(* IEC 61131-3 sources: beeguard/archive, 2 files *)

(* ---- analog.st ---- *)
FUNCTION_BLOCK AOI_CM_AIN
VAR_INPUT
	IN_IOH: BOOL;
	IN_INH1: DINT;
	IN_OVR: BOOL;
	IN_UNR: BOOL;
	IN_RAW: REAL;
	CMD_ALM_RES: BOOL;
	IN_CLOCK: DT;	// CURRENT DATE AND TIME, PASSED TO THE ALARMS FOR TIME STAMPS
END_VAR
VAR_INPUT PERSISTENT RETAIN
	CFG_EN: BOOL;
	CFG_RU_MAX: DINT;
	CFG_RU_MIN: DINT;
	CFG_EU_MAX: REAL;
	CFG_EU_MIN: REAL;
	CFG_HIHI_SP: REAL;
	CFG_HI_SP: REAL;
	CFG_LO_SP: REAL;
	CFG_LOLO_SP: REAL;
	CFG_FRZN_SP: REAL;
	CFG_DEC_PT: DINT;
	CFG_DESC: STRING;
	CFG_DEV_TYPE: DINT;
	CFG_EID: STRING;
	CFG_EN_ALM_HI: BOOL;
	CFG_EN_ALM_HIHI: BOOL;
	CFG_EN_ALM_IOH: BOOL;
	CFG_EN_ALM_LO: BOOL;
	CFG_EN_ALM_LOLO: BOOL;
	CFG_EN_ALM_OOR: BOOL;
	CFG_EN_ALM_FRZN: BOOL;
	CFG_EN_IOH: BOOL;
	CFG_EN_OOR: BOOL;
	CFG_EN_SCL: BOOL;
	CFG_EN_TOT: BOOL;
	CFG_EN_FRZN: BOOL;
	CFG_HI_DT: DINT;
	CFG_HIHI_DT: DINT;
	CFG_LO_DT: DINT;
	CFG_LOLO_DT: DINT;
	CFG_OOR_DT: DINT;
	CFG_FRZN_DT: DINT;
	CFG_SCL_TYP: DINT;
	CFG_UNITS: STRING;
	SIM: BOOL;
	CFG_TMR_DISABLE_SIM: BOOL;
END_VAR
VAR_IN_OUT
	ALMD_HIHI: BG_ALM_DIG;
	ALMD_HI: BG_ALM_DIG;
	ALMD_LO: BG_ALM_DIG;
	ALMD_LOLO: BG_ALM_DIG;
	ALMD_OOR: BG_ALM_DIG;
	ALMD_IOH: BG_ALM_DIG;
	ALMD_FRZN: BG_ALM_DIG;
END_VAR
VAR_OUTPUT
	STS_RDY2GO: BOOL;
	VAL_ACT: REAL;
	ALM_HIHI: BOOL;
	ALM_HI: BOOL;
	ALM_LO: BOOL;
	ALM_LOLO: BOOL;
	ALM_OOR: BOOL;
	ALM_IOH: BOOL;
	ALM_FRZN: BOOL;
	STS_HIHI: BOOL;
	STS_HI: BOOL;
	STS_LO: BOOL;
	STS_LOLO: BOOL;
	STS_OOR: BOOL;
	STS_IOH: BOOL;
	STS_FRZN: BOOL;
	CFG_VERSION: REAL;
	STS_ALM_ANY: BOOL;
	STS_ALM_ANY_UNACK: BOOL;
	ALM_ANY: BOOL;
	VAL_S: DINT;
END_VAR
VAR
	SIM_ONS: R_TRIG;
	WRK_B0: BOOL;
	WRK_B1: BOOL;
	WRK_ONS: ARRAY[0..15] OF R_TRIG;
	WRK_R: ARRAY[0..6] OF REAL;
	WRK_T: ARRAY[0..7] OF TON;
END_VAR

(*===========================================================================
AOI: CM_AIN
Date Last Updated: 5-27-2024
===========================================================================*)
//CFG_VERSION:= 1.0; // ORIGINAL
//CFG_VERSION := 2.0; //ADDED THE DIGITAL ALARM FUNCTION BLOCK
//CFG_VERSION := 2.1; //ADDED FRONZEN DATA ALARM LOGIC
//CFG_VERSION := 2.2; //DIGITAL ALARM 3.0: ACK+RESET, CLOCK, INHIBIT = SUPPRESS, SINGLE ON-DELAY, IOH INHIBIT ON BIT 6
CFG_VERSION := 2.3; //USES BG_ALM_DIG 3.1 NAMES; CLOCK INPUT RENAMED IN_CLOCK
(*===========================================================================
RETURN IF DISABLED  - If Module is Disabled, Scan One Last Time for Cleanup, Then Return
===========================================================================*)
IF NOT(CFG_EN) THEN
	WRK_ONS[1].CLK := TRUE;
	IF WRK_ONS[1].Q THEN
		WRK_B1 := TRUE;
	END_IF
	IF NOT(WRK_B1) THEN
		JMP EXIT_AOI_CM_AIN;
	END_IF
ELSE
	WRK_B1 := FALSE;
	WRK_ONS[1].CLK := FALSE;
END_IF

(*===========================================================================
SETUP - Clean up the Config: Enable Alarming depending on what Inputs are Confirmed in the System.
===========================================================================*)
IF NOT(CFG_EN_IOH) THEN
	CFG_EN_ALM_IOH := FALSE;
END_IF
IF NOT(CFG_EN_OOR) THEN
	CFG_EN_ALM_OOR := FALSE;
END_IF
IF NOT(CFG_EN_FRZN) THEN
	CFG_EN_ALM_FRZN := FALSE;
END_IF
(*===========================================================================
SETUP - Prevent wire-framing in HMI during start up (this prevents dividing by zero).
===========================================================================*)
IF CFG_EU_MAX = 0.0 THEN
	CFG_EU_MAX := 100;
END_IF

(*===========================================================================
TIMER PRESETS - Check and correct for invalid Timer Preset values
===========================================================================*)
WRK_T[1].PT := DINT_TO_TIME(ABS(CFG_HIHI_DT)*1000);
WRK_T[2].PT := DINT_TO_TIME(ABS(CFG_HI_DT)*1000);
WRK_T[3].PT := DINT_TO_TIME(ABS(CFG_LO_DT)*1000);
WRK_T[4].PT := DINT_TO_TIME(ABS(CFG_LOLO_DT)*1000);
WRK_T[5].PT := DINT_TO_TIME(ABS(CFG_OOR_DT)*1000);
WRK_T[7].PT := DINT_TO_TIME(ABS(CFG_FRZN_DT)*1000);

(*===========================================================================
COMMANDS - Latch Internal Work Bit To Clear All Alarms
===========================================================================*)
SIM_ONS.CLK := SIM;
IF CMD_ALM_RES OR (SIM_ONS.Q) THEN
	WRK_B0 := TRUE;
	CMD_ALM_RES := FALSE;
END_IF

(*===========================================================================
STATUS - I/O Health
===========================================================================*)
IF (CFG_EN_IOH AND IN_IOH) OR (NOT(CFG_EN_IOH)) OR (SIM) THEN
	STS_IOH := TRUE;
ELSE
	STS_IOH := FALSE;
END_IF

(*===========================================================================
STATUS - I/O Health
===========================================================================*)
IF (CFG_EN_OOR) AND (IN_OVR OR IN_UNR) THEN
	STS_OOR := TRUE;
ELSE
	STS_OOR := FALSE;
END_IF

(*===========================================================================
STATUS  - CM Ready to Go
CM is Ready to Go if it is Enabled, it's HOA(s) are in the Auto position and Interlocks are met.
NOTE: Not all conditions may exist for a given CM Cla
===========================================================================*)
IF (CFG_EN AND STS_IOH) THEN
	STS_RDY2GO := TRUE;
ELSE
	STS_RDY2GO := FALSE;
END_IF

(*===========================================================================
ALARMS HIHI - Determine HIHI Alarm if Alarms are Enabled.  If an Alarm is already
present when it is Disabled becomes it will stay TRUE.
===========================================================================*)
IF (VAL_ACT > CFG_HIHI_SP) THEN
	WRK_T[1](IN := TRUE);
	IF WRK_T[1].Q THEN
		STS_HIHI := TRUE;
		IF NOT(IN_INH1.0) AND CFG_EN_ALM_HIHI THEN
			ALM_HIHI := TRUE;
		ELSE
			ALM_HIHI := FALSE;
		END_IF
	ELSE
		STS_HIHI := FALSE;
	END_IF
ELSE
	STS_HIHI := FALSE;
	ALM_HIHI := FALSE;
	WRK_T[1](IN := FALSE);
END_IF

// INHIBIT SUPPRESSES THE ALARM INSTEAD OF RETURNING IT TO NORMAL. WRK_T[1] IS THE ONLY ON-DELAY.
ALMD_HIHI(IN_SIGNAL := CFG_EN_ALM_HIHI AND STS_HIHI, CMD_PG_SUPPRESS := IN_INH1.0, CMD_PG_UNSUPPRESS := NOT(IN_INH1.0),
	CFG_ACK_REQ := TRUE, CFG_LATCH := TRUE, CFG_ON_DELAY_MS := 0, IN_CLOCK := IN_CLOCK);

IF WRK_B0 THEN
	 WRK_ONS[5].CLK := TRUE;
	 IF WRK_ONS[5].Q THEN
		 ALMD_HIHI.CMD_OP_ACK := TRUE;
		 ALMD_HIHI.CMD_OP_RESET := TRUE;
	 END_IF
ELSE
	WRK_ONS[5].CLK := FALSE;
END_IF

(*===========================================================================
ALARMS HI - Determine HI Alarm if Alarms are Enabled.  If an Alarm is already
present when it is Disabled becomes it will stay TRUE.
===========================================================================*)
IF (VAL_ACT > CFG_HI_SP) THEN
	WRK_T[2](IN := TRUE);
	IF WRK_T[2].Q THEN
		STS_HI := TRUE;
		IF NOT(IN_INH1.1) AND CFG_EN_ALM_HI THEN
			ALM_HI := TRUE;
		ELSE
			ALM_HI := FALSE;
		END_IF
	ELSE
		STS_HI := FALSE;
	END_IF
ELSE
	STS_HI := FALSE;
	ALM_HI := FALSE;
	WRK_T[2](IN := FALSE);
END_IF

ALMD_HI(IN_SIGNAL := CFG_EN_ALM_HI AND STS_HI, CMD_PG_SUPPRESS := IN_INH1.1, CMD_PG_UNSUPPRESS := NOT(IN_INH1.1),
	CFG_ACK_REQ := TRUE, CFG_LATCH := TRUE, CFG_ON_DELAY_MS := 0, IN_CLOCK := IN_CLOCK);

IF WRK_B0 THEN
	 WRK_ONS[7].CLK := TRUE;
	 IF WRK_ONS[7].Q THEN
		 ALMD_HI.CMD_OP_ACK := TRUE;
		 ALMD_HI.CMD_OP_RESET := TRUE;
	 END_IF
ELSE
	WRK_ONS[7].CLK := FALSE;
END_IF

(*===========================================================================
ALARMS LO - Determine LO Alarm if Alarms are Enabled.  If an Alarm is already
present when it is Disabled becomes it will stay TRUE.
===========================================================================*)
IF (VAL_ACT < CFG_LO_SP) THEN
	WRK_T[3](IN := TRUE);
	IF WRK_T[3].Q THEN
		STS_LO := TRUE;
		IF NOT(IN_INH1.2) AND CFG_EN_ALM_LO THEN
			ALM_LO := TRUE;
		ELSE
			ALM_LO := FALSE;
		END_IF
	ELSE
		STS_LO := FALSE;
	END_IF
ELSE
	STS_LO := FALSE;
	ALM_LO := FALSE;
	WRK_T[3](IN := FALSE);
END_IF

ALMD_LO(IN_SIGNAL := CFG_EN_ALM_LO AND STS_LO, CMD_PG_SUPPRESS := IN_INH1.2, CMD_PG_UNSUPPRESS := NOT(IN_INH1.2),
	CFG_ACK_REQ := TRUE, CFG_LATCH := TRUE, CFG_ON_DELAY_MS := 0, IN_CLOCK := IN_CLOCK);

IF WRK_B0 THEN
	 WRK_ONS[9].CLK := TRUE;
	 IF WRK_ONS[9].Q THEN
		 ALMD_LO.CMD_OP_ACK := TRUE;
		 ALMD_LO.CMD_OP_RESET := TRUE;
	 END_IF
ELSE
	WRK_ONS[9].CLK := FALSE;
END_IF

(*===========================================================================
ALARMS LOLO - Determine LOLO Alarm if Alarms are Enabled.  If an Alarm is already
present when it is Disabled becomes it will stay TRUE.
===========================================================================*)
IF (VAL_ACT < CFG_LOLO_SP) THEN
	WRK_T[4](IN := TRUE);
	IF WRK_T[4].Q THEN
		STS_LOLO := TRUE;
		IF NOT(IN_INH1.3) AND CFG_EN_ALM_LOLO THEN
			ALM_LOLO := TRUE;
		ELSE
			ALM_LOLO := FALSE;
		END_IF
	ELSE
		STS_LOLO := FALSE;
	END_IF
ELSE
	STS_LOLO := FALSE;
	ALM_LOLO := FALSE;
	WRK_T[4](IN := FALSE);
END_IF

ALMD_LOLO(IN_SIGNAL := CFG_EN_ALM_LOLO AND STS_LOLO, CMD_PG_SUPPRESS := IN_INH1.3, CMD_PG_UNSUPPRESS := NOT(IN_INH1.3),
	CFG_ACK_REQ := TRUE, CFG_LATCH := TRUE, CFG_ON_DELAY_MS := 0, IN_CLOCK := IN_CLOCK);

IF WRK_B0 THEN
	 WRK_ONS[11].CLK := TRUE;
	 IF WRK_ONS[11].Q THEN
		 ALMD_LOLO.CMD_OP_ACK := TRUE;
		 ALMD_LOLO.CMD_OP_RESET := TRUE;
	 END_IF
ELSE
	WRK_ONS[11].CLK := FALSE;
END_IF

(*===========================================================================
ALARMS - Out of Range
===========================================================================*)
IF (CFG_EN_ALM_OOR AND STS_OOR) THEN
	WRK_T[5](IN := TRUE);
	IF WRK_T[5].Q THEN
		//STS_OOR := TRUE; SEE LINE 35
		IF NOT(IN_INH1.4) THEN
			ALM_OOR := TRUE;
		ELSE
			ALM_OOR := FALSE;
		END_IF
	END_IF
ELSE
	ALM_OOR := FALSE;
	WRK_T[5](IN := FALSE);
END_IF

ALMD_OOR(IN_SIGNAL := CFG_EN_ALM_OOR AND STS_OOR AND WRK_T[5].Q, CMD_PG_SUPPRESS := IN_INH1.4, CMD_PG_UNSUPPRESS := NOT(IN_INH1.4),
	CFG_ACK_REQ := TRUE, CFG_LATCH := TRUE, CFG_ON_DELAY_MS := 0, IN_CLOCK := IN_CLOCK);

IF WRK_B0 THEN
	 WRK_ONS[13].CLK := TRUE;
	 IF WRK_ONS[13].Q THEN
		 ALMD_OOR.CMD_OP_ACK := TRUE;
		 ALMD_OOR.CMD_OP_RESET := TRUE;
	 END_IF
ELSE
	WRK_ONS[13].CLK := FALSE;
END_IF

(*===========================================================================
ALARMS - FROZEN VALUE
===========================================================================*)
IF (VAL_ACT = CFG_FRZN_SP) THEN
	STS_FRZN := TRUE;
ELSE
	STS_FRZN := FALSE;
END_IF

IF (CFG_EN_ALM_FRZN AND STS_FRZN) THEN
	WRK_T[7](IN := TRUE);
	IF WRK_T[7].Q THEN
		//STS_FRZN := TRUE; SEE LINE 35
		IF NOT(IN_INH1.5)THEN
			ALM_FRZN := TRUE;
		ELSE
			ALM_FRZN := FALSE;
		END_IF
	END_IF
ELSE
	ALM_FRZN := FALSE;
	WRK_T[7](IN := FALSE);
END_IF

IF WRK_T[7].ET > T#0S OR CFG_EN_ALM_FRZN THEN
	CFG_FRZN_SP := VAL_ACT;
END_IF

// CFG_FRZN_DT IS NOW THE ONLY FROZEN DELAY (THE EXTRA 60 S IN THE ALARM BLOCK WAS REMOVED).
ALMD_FRZN(IN_SIGNAL := CFG_EN_ALM_FRZN AND STS_FRZN AND WRK_T[7].Q, CMD_PG_SUPPRESS := IN_INH1.5, CMD_PG_UNSUPPRESS := NOT(IN_INH1.5),
	CFG_ACK_REQ := TRUE, CFG_LATCH := TRUE, CFG_ON_DELAY_MS := 0, IN_CLOCK := IN_CLOCK);

IF WRK_B0 THEN
	 WRK_ONS[14].CLK := TRUE;
	 IF WRK_ONS[14].Q THEN
		 ALMD_FRZN.CMD_OP_ACK := TRUE;
		 ALMD_FRZN.CMD_OP_RESET := TRUE;
	 END_IF
ELSE
	WRK_ONS[14].CLK := FALSE;
END_IF

(*===========================================================================
ALARM - I/O Health (Includes Module Health, Channel Calibration Fault, or Channel Fault Alarms)
===========================================================================*)
// I/O HEALTH HAS ITS OWN INHIBIT BIT 6 (IT SHARED BIT 5 WITH FROZEN VALUE).
// IT HAS NO OTHER DELAY, SO IT KEEPS THE 1 S ON-DELAY IN THE ALARM BLOCK.
IF CFG_EN_ALM_IOH AND NOT(STS_IOH) AND NOT(IN_INH1.6) THEN
	ALM_IOH := TRUE;
ELSE
	ALM_IOH := FALSE;
END_IF

ALMD_IOH(IN_SIGNAL := CFG_EN_ALM_IOH AND NOT(STS_IOH), CMD_PG_SUPPRESS := IN_INH1.6, CMD_PG_UNSUPPRESS := NOT(IN_INH1.6),
	CFG_ACK_REQ := TRUE, CFG_LATCH := TRUE, CFG_ON_DELAY_MS := 1000, IN_CLOCK := IN_CLOCK);

IF WRK_B0 THEN
	 WRK_ONS[15].CLK := TRUE;
	 IF WRK_ONS[15].Q THEN
		 ALMD_IOH.CMD_OP_ACK := TRUE;
		 ALMD_IOH.CMD_OP_RESET := TRUE;
	 END_IF
ELSE
	WRK_ONS[15].CLK := FALSE;
END_IF

(*===========================================================================
ALARMS - Any Alarm
===========================================================================*)
IF ALM_HIHI OR ALM_HI OR ALM_LO OR ALM_LOLO OR ALM_OOR OR ALM_IOH OR ALM_FRZN THEN
	ALM_ANY := TRUE;
	STS_ALM_ANY := TRUE;
ELSE
	ALM_ANY := FALSE;
	STS_ALM_ANY := FALSE;
END_IF

(*===========================================================================
ALARMS - Check to see if there are any unacknowledged alarms, including latched
alarms whose condition has already cleared.
===========================================================================*)
IF ALMD_HIHI.STS_UNACKED OR ALMD_HI.STS_UNACKED OR ALMD_LO.STS_UNACKED OR ALMD_LOLO.STS_UNACKED OR ALMD_OOR.STS_UNACKED OR ALMD_IOH.STS_UNACKED OR ALMD_FRZN.STS_UNACKED THEN
	STS_ALM_ANY_UNACK := TRUE;
ELSE
	STS_ALM_ANY_UNACK := FALSE;
END_IF

(*===========================================================================
VALUES - State (HMI Color)
0 = Normal
1 = In Alarm
2 = Disabled
===========================================================================*)
IF NOT ALM_ANY THEN
	VAL_S := 0;
END_IF
IF ALM_ANY AND STS_ALM_ANY_UNACK THEN
	VAL_S := 1;
END_IF
IF ALM_ANY AND NOT STS_ALM_ANY_UNACK THEN
	VAL_S := 3;
END_IF

(*===========================================================================
VALUES - Actual Value
===========================================================================*)
IF CFG_EN_SCL THEN
	// SCALING CONFIGURATION
	IF CFG_SCL_TYP <> 1 AND CFG_SCL_TYP <> 2 THEN
		CFG_SCL_TYP := 1;
	END_IF
	IF CFG_RU_MAX = 0 AND CFG_RU_MIN = 0 THEN
		CFG_RU_MAX := 20;
		CFG_RU_MIN := 4;
	END_IF
	IF CFG_EU_MAX = 0 THEN
		CFG_EU_MAX := 1;
	END_IF
	IF CFG_RU_MAX = 0 THEN
		CFG_RU_MAX := 1;
	END_IF
	// LINEAR SCALING
	IF CFG_SCL_TYP = 1 THEN
		IF CFG_RU_MAX > CFG_RU_MIN THEN
			WRK_R[4] := (IN_RAW - DINT_TO_REAL(CFG_RU_MIN))/DINT_TO_REAL(CFG_RU_MAX - CFG_RU_MIN) * (CFG_EU_MAX-CFG_EU_MIN)+CFG_EU_MIN;
		END_IF
	END_IF
	// NON-LINEAR SCALING CONFIGURATION
	IF CFG_SCL_TYP = 2 THEN
		IF CFG_EU_MIN >= 0 THEN
			WRK_R[1] := LREAL_TO_REAL(EXPT(CFG_EU_MIN, 2));
		END_IF
		IF CFG_EU_MIN < 0 THEN
			WRK_R[1] := LREAL_TO_REAL(-1.0*EXPT(CFG_EU_MIN, 2));
		END_IF
		IF CFG_EU_MAX >= 0 THEN
			WRK_R[2] := LREAL_TO_REAL(EXPT(CFG_EU_MAX, 2));
		END_IF
		IF CFG_EU_MAX < 0 THEN
			WRK_R[2] := LREAL_TO_REAL(-1.0*EXPT(CFG_EU_MAX, 2));
		END_IF
		// NON-LINEAR SCALING
		IF CFG_RU_MAX > CFG_RU_MIN THEN
			WRK_R[3] := (IN_RAW - DINT_TO_REAL(CFG_RU_MIN))* (WRK_R[2] - WRK_R[1])/ DINT_TO_REAL(CFG_RU_MAX-CFG_RU_MIN)+ WRK_R[1];
		END_IF
		IF WRK_R[3] >= 0 THEN
			WRK_R[4] := SQRT(WRK_R[3]);
		END_IF
		IF WRK_R[3] < 0 THEN
			WRK_R[4] := -1.0 * SQRT(WRK_R[3]);
		END_IF
	END_IF
END_IF

IF NOT CFG_EN_SCL THEN
	WRK_R[4] := IN_RAW;
END_IF

VAL_ACT := WRK_R[4];

IF SIM THEN
	VAL_ACT := WRK_R[5];
END_IF

(*===========================================================================
SIM - Don't let the SIM bit stay on for more than 24 hours.
ADDED - TIMER BYPASS: NOTE SIM IS FOREVER!!!!
===========================================================================*)
IF SIM AND NOT CFG_TMR_DISABLE_SIM THEN
	WRK_T[6](IN := TRUE, PT := T#1440000MS);
	IF WRK_T[6].Q THEN
		SIM := FALSE;
	END_IF
ELSE
	WRK_T[6](IN := FALSE);
END_IF

(*===========================================================================
Unlatch Alarms Reset Bit
===========================================================================*)
IF WRK_B0 THEN
	WRK_B0 := FALSE;
END_IF

(*===========================================================================
CM DISABLED - Set Conditions Upon Entering Disabled State
===========================================================================*)
IF WRK_B1 THEN
	WRK_B0 := FALSE;
	VAL_S := 3;
	SIM := FALSE;
END_IF

(*===========================================================================
Exit AOI
===========================================================================*)
EXIT_AOI_CM_AIN:

END_FUNCTION_BLOCK

(* ---- digital_alarm_v2.st ---- *)
FUNCTION_BLOCK AOI_CM_ALMD
(*==========================================================================
v2.0 of the digital alarm block, kept as a historical record. It was replaced
by v3.0, now BG_ALM_DIG in reference/digital_alarm.st. The code below is the
original v2.0 and is not maintained; its block and parameter names are the
originals and are not used anywhere else.

WHAT v2.0 SET OUT TO DO
	Raise an alarm from one BOOL signal (IN), optionally inverted (CONDITION =
	TRUE), with an optional minimum time in alarm (MINDURATIONPRE, ms), an
	optional acknowledge requirement (ACKREQUIRED) and optional latching until
	a reset (LATCHED). Operator requests (OPER*) and logic requests (PROG*)
	were meant to acknowledge, reset, take the alarm out of service, suppress
	it and shelve it, the last three corresponding to ISA-18.2 states H, G and
	F. Outputs report whether the alarm is in alarm and acknowledged, how often
	it has activated, and when (INALARMTIME, ACKTIME, RETONORMALTIME, ...).
	STATE reported ISA-18.2 states A to D: 0 normal, 1 in alarm unacknowledged,
	2 in alarm acknowledged, 3 back to normal unacknowledged.

WHY IT WAS REPLACED - DEFECTS FOUND IN REVIEW
	- INALARM := MINDURATION.Q is overwritten by INALARM := IN, so the minimum
	  duration has no effect on INALARM.
	- CONDITION only inverts INALARM; the state transitions test the raw IN.
	- STATE is recomputed from INALARM/ACKED every scan, so the block does not
	  remember its state and latching does not hold.
	- Latched states 1 and 2 clear on NOT IN, and state 3 returns to NORMAL with
	  no acknowledgement.
	- A reset sets ACKED, and the acknowledge test in the same scan then moves
	  the alarm to state 2 (INALARM TRUE). The non-latched RTN path has the same
	  problem going from state 3 to state 2.
	- Suppress writes to the disable inputs, and the command resets at the end
	  cancel opposing pairs, so suppress and disable are mixed up.
	- Shelving is declared but not implemented: OPERSHELVE, OPERUNSHELVE,
	  PROGSHELVE, PROGUNSHELVE, MAXSHELVEDURATION and SEVERITY are never read;
	  SHELVED, SUPPRESSED, DIABLED, ALARMCOUNT, INALARMUNACK and INSTRUCTFAULT
	  are never written.
	- PROGTIME is overwritten from M_TX; the time stamps are TIME durations from
	  OSCAT M_TX, not date-times, and ACKTIME is the "time high", not the ack time.
	- Only OPERACK and PROGACK are cleared; PROG* commands are level, not edge.
	- MINDURATIONACC is an INT and overflows after 32.767 s. The timer
	  instances are declared as outputs.
	- Typos: DIABLED, OPERDISBLE, PROGUNSUPRESS, USEPROTIME (duplicate of USEPROGTIME).
==========================================================================*)
VAR_INPUT
	(* INPUTS *)
	ENABLEIN: BOOL;
	IN: BOOL; //DIGITAL ALARM
	INFAULT: BOOL;
	CONDITION: BOOL; //INVERT INPUT SIGNAL
	ACKREQUIRED: BOOL; // ACKKNOWLEDGE REQUIREMENT
	LATCHED: BOOL;	//LATCH REQUIREMENT
	MINDURATIONPRE: DINT;

	OPERACK: BOOL;
	OPERRESET: BOOL;
	OPERDISBLE: BOOL;
	OPERENABLE: BOOL;
	OPERSUPPRESS: BOOL;
	OPERUNSUPPRESS: BOOL;
	OPERSHELVE: BOOL;
	OPERUNSHELVE: BOOL;

	PROGACK: BOOL;
	PROGRESET: BOOL;
	PROGDISABLE: BOOL;
	PROGENABLE: BOOL;
	PROGSUPPRESS: BOOL;
	PROGUNSUPRESS: BOOL;
	PROGSHELVE: BOOL;
	PROGUNSHELVE: BOOL;

	ALARMCOUNTRESET: BOOL;
	USEPROGTIME: BOOL;
	SEVERITY: DINT;
	MAXSHELVEDURATION: DINT;

	USEPROTIME: BOOL;
	PROGTIME: TIME;
END_VAR
VAR_OUTPUT
	ENABLEOUT: BOOL;
	INALARM: BOOL;
	ACKED: BOOL;
	INALARMUNACK: BOOL;
	SUPPRESSED: BOOL;
	SHELVED: BOOL;
	DIABLED: BOOL;
	INSTRUCTFAULT: BOOL;
	ALARMCOUNT: DINT;

	INALARMTIME: TIME;
	ACKTIME: TIME;
	RETONORMALTIME: TIME;
	ALARMCOUNTRESETTIME: TIME;

	SHELVETIME: TIME;
	UNSHELVETIME: TIME;

	STATE: DINT;
	STATUS: DINT;

	MINDURATIONACC: INT;
	INFAULTED: BOOL;

	MINDURATION: TON;
	ALARMTIME: OSCAT_BASIC.M_TX;
	CFG_VERSION: REAL;
END_VAR

(*==========================================================================
Sets the Version of the Control Module on the HMI and in the Program.
==========================================================================
Date Last Updated: 5-27-2024
===========================================================================*)
//CFG_VERSION:= 1.0; // ORIGINAL
CFG_VERSION := 2.0; //ADDED AOI_CM_ALMD FUNCTION BLOCK
MINDURATION(IN:=IN, PT:=DINT_TO_TIME(MINDURATIONPRE));
MINDURATIONACC := TIME_TO_INT(MINDURATION.ET);
INALARM := MINDURATION.Q;
ALARMTIME(in:= IN,rst:=ALARMCOUNTRESET);

IF NOT CONDITION THEN
	INALARM := IN;
ELSE
	INALARM := NOT IN;
END_IF

IF OPERSUPPRESS THEN
	OPERDISBLE := TRUE;
	OPERENABLE := FALSE;
END_IF

IF OPERUNSUPPRESS THEN
	OPERDISBLE := FALSE;
	OPERENABLE := TRUE;
END_IF

IF PROGSUPPRESS THEN
	PROGDISABLE := TRUE;
	PROGENABLE := FALSE;
END_IF

IF PROGUNSUPRESS THEN
	PROGDISABLE := FALSE;
	PROGENABLE := TRUE;
END_IF

IF ENABLEIN AND NOT (OPERSUPPRESS OR PROGSUPPRESS) THEN
	ENABLEOUT := TRUE;
ELSE
	ENABLEOUT := FALSE;
END_IF

IF ACKREQUIRED THEN
	IF NOT INALARM AND ACKED THEN
		STATE := 0;
	ELSIF INALARM AND NOT ACKED THEN
		STATE := 1;
	ELSIF INALARM AND ACKED THEN
		STATE := 2;
	ELSIF NOT INALARM AND NOT ACKED THEN
		STATE := 3;
	ELSE
		//DO NOTHING
	END_IF

	IF LATCHED THEN
		CASE STATE OF
		0:
			IF IN AND MINDURATION.Q THEN
				STATE := 1;
				INALARM := TRUE;
				ACKED := FALSE;
			END_IF
		1:
			IF NOT IN OR OPERRESET OR PROGRESET THEN
				STATE := 0;
				INALARM := FALSE;
				ACKED := TRUE;
			END_IF

			IF ACKED OR PROGACK OR OPERACK THEN
				STATE := 2;
				INALARM := TRUE;
				ACKED := TRUE;
			END_IF
		2:
			IF NOT IN OR OPERRESET OR PROGRESET THEN
				STATE := 0;
				INALARM := FALSE;
				ACKED := TRUE;
			END_IF
		3:
			STATE := 0;
		END_CASE

	ELSE
		CASE STATE OF
		0:
			IF IN AND MINDURATION.Q THEN
				STATE := 1;
				INALARM := TRUE;
				ACKED := FALSE;
			END_IF
		1:
			IF NOT IN THEN
				STATE := 3;
				INALARM := FALSE;
				ACKED := FALSE;
			END_IF

			IF ACKED OR PROGACK OR OPERACK THEN
				STATE := 2;
				INALARM := TRUE;
				ACKED := TRUE;
			END_IF
		2:
			IF NOT IN THEN
				STATE := 0;
				INALARM := FALSE;
				ACKED := TRUE;
			END_IF
		3:
			IF ACKED OR OPERACK OR PROGACK THEN
				STATE := 0;
				INALARM := FALSE;
				ACKED := TRUE;
			END_IF

			IF IN AND MINDURATION.Q THEN
				STATE := 1;
				INALARM := TRUE;
				ACKED := FALSE;
			END_IF
		END_CASE
	END_IF
END_IF

IF NOT ACKREQUIRED THEN
	IF NOT INALARM THEN
		STATE := 0;
	ELSIF INALARM THEN
		STATE := 1;
	ELSE
		//DO NOTHING
	END_IF

	IF  LATCHED THEN
		CASE STATE OF
			0:
				IF IN AND MINDURATION.Q THEN
					STATE := 1;
					INALARM := TRUE;
				END_IF
			1:
				IF NOT IN OR OPERRESET OR PROGRESET THEN
					STATE := 0;
					INALARM := FALSE;
				END_IF
		END_CASE
	ELSE
		CASE STATE OF
			0:
				IF IN AND MINDURATION.Q THEN
					STATE := 1;
					INALARM := TRUE;
				END_IF
			1:
				IF NOT IN THEN
					STATE := 0;
					INALARM := FALSE;
				END_IF
		END_CASE
	END_IF
END_IF

//OUTPUT UPDATES
PROGTIME := ALARMTIME.ET;
ACKTIME := ALARMTIME.TH;
RETONORMALTIME := ALARMTIME.TL;

IF PROGSUPPRESS THEN
	PROGUNSUPRESS := FALSE;
END_IF

IF OPERSUPPRESS THEN
	OPERUNSUPPRESS := FALSE;
END_IF

IF PROGUNSUPRESS THEN
	PROGSUPPRESS := FALSE;
END_IF

IF OPERUNSUPPRESS THEN
	OPERSUPPRESS := FALSE;
END_IF

IF INALARM AND (PROGSUPPRESS OR OPERSUPPRESS) THEN
	INALARM := FALSE;
END_IF

IF INALARM AND (PROGUNSUPRESS OR OPERUNSUPPRESS) THEN
	INALARM := TRUE;
END_IF

IF INFAULT THEN
	STATUS.1 := TRUE;
ELSE
	STATUS.1 := FALSE;
END_IF

//COMMAND RESETS
OPERACK := FALSE;
PROGACK := FALSE;

END_FUNCTION_BLOCK
